TYPE s_str_alarmList :
STRUCT
	var_alarmLevel : STRING;
	var_alarmName : WSTRING;
	var_alarmMassge : WSTRING;
	var_alarmTime : STRING;
	var_alarmCode1 : eP_alarmCode;
	var_alarmCode2 : STRING;
	
END_STRUCT
END_TYPE

(* stored: Version 1.1.0.1, ProductVersion 3.1.4024.11
   DUT s_str_alarmList: Id {d5551d26-3c37-4c79-a029-3cfd3ac0f6b6} *)
